(* CoDeSys 2.3 export: STATE_MACHINES.EXP *)

(* Global variable list: State_Machines *)
VAR_GLOBAL
	stMachine_s16				: INT		:= 0;		(*	machine state 	*)
	stStartlock_b8				: BOOL; 				(* No HW problems detected at start, if TRUE *)
	stStartAppl_b8				: BOOL;				(* Application Start condition OK, if TRUE *)
END_VAR

VAR_GLOBAL CONSTANT

(*************************************************************************************************)
	DEACTIVATED				:	INT	:=	0;
	ACTIVATED				:	INT	:=	1;

END_VAR
